(* IEC 61131-3 sources: CodesysTest/alpha/export/FBs/Components/Cylinders/FB_Cylinder.pou, 1 file *)

(* ---- FB_Cylinder.pou.st ---- *)
(*#-#-#-#-#-#-#-#-#-#---Declaration---#-#-#-#-#-#-#-#-#-#-#-#-#*)

FUNCTION_BLOCK FB_Cylinder IMPLEMENTS ICylinder
VAR_INPUT
    mode : DEVICE_MODES;
END_VAR
VAR_OUTPUT
    extendedStatus : BOOL;
    retractedStatus : BOOL;
    extendOutput : BOOL;
    retractOutput : BOOL;
END_VAR
VAR
END_VAR
(*#-#-#-#-#-#-#-#-#-#---Implementation---#-#-#-#-#-#-#-#-#-#-#-#-#*)
